FUNCTION_BLOCK FB_CTU_AI (* Up counter (INT) *)
  (* Standard: 61499-1; Description: Copyright (c) 2023 Martin Erich Jobst This program and the accompanying materials are made available under the terms of the Eclipse Public License 2.0 which is available at https://www.eclipse.org/legal/epl-2.0/ SPDX-License-Identifier: EPL-2.0 *)
  (* Version 3.0, 2025-04-14, Patrick Aigner, changed package *)
  (* Version 1.0, 2023-04-28, Martin Jobst *)
  PACKAGE adapter::iec61131::counters;
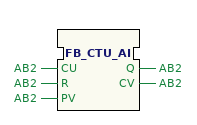
  SOCKETS
    CU : adapter::types::bidirectional::AB2; (* Count up *)
    R : adapter::types::bidirectional::AB2; (* Reset *)
    PV : adapter::types::bidirectional::AB2; (* Preset value *)
  END_SOCKETS
  PLUGS
    Q : adapter::types::bidirectional::AB2; (* Output *)
    CV : adapter::types::bidirectional::AB2; (* Count value *)
  END_PLUGS
  EC_STATES
    REQ : REQ -> CNF;
  END_STATES
  ALGORITHM REQ IN ST:
IF R THEN
  CV := 0;
ELSIF CU AND CV < 32767 THEN
  CV := CV + 1;
END_IF;
Q := CV>= PV;
  END_ALGORITHM
END_FUNCTION_BLOCK
